% RSLogix 500 project XLT_EXP_TOP.RSS, saved by version 11.00.00.00 %
PROJECT "LINCETOP"    % processor: MicroLogix 1400 %

PROGRAM FILES
  LAD 2 "MAIN"  15 rungs  % Main Program Routine %
  LAD 70 "OFFSETS"  13 rungs
  LAD 88 "TIMESWITCH"  2 rungs
  LAD 89 "SECONDS"  2 rungs
  LAD 90 "HSC"  9 rungs
  LAD 99 "HMI SET"  3 rungs
  LAD 100 "STI"  32 rungs
  LAD 102 "SPEED"  6 rungs
  LAD 104 "P ADJUST"  8 rungs
  LAD 110 "SHIFT"  11 rungs
  LAD 120 "XFER IN"  3 rungs
  LAD 121 "NOTUSED4"  7 rungs
  LAD 122 "PARTDETECT"  9 rungs
  LAD 123 "OPTICWIDTH"  8 rungs
  LAD 124 "PART GAP"  8 rungs
  LAD 125 "NOTUSED2"  4 rungs
  LAD 126 "ALIGNLOAD"  15 rungs
  LAD 127 "NOTUSED"  3 rungs
  LAD 128 "NOTUSED3"  12 rungs
  LAD 130 "INS 5 TRIG"  30 rungs
  LAD 131 "INS 5 RSLT"  29 rungs
  LAD 140 "INS 6 TRIG"  30 rungs
  LAD 141 "INS 6 RSLT"  30 rungs
  LAD 170 "PASSBLOW"  14 rungs
  LAD 180 "RECERK"  9 rungs
  LAD 200 "PRODRATE"  6 rungs
  LAD 230 "HMI GET"  1 rungs

DATA FILES
  O0 OUTPUT  6 elements
  I1 INPUT  8 elements
  S2 STATUS  66 elements
  B3 BINARY  14 elements
  T4 TIMER  40 elements
  C5 COUNTER  1 elements
  R6 CONTROL  30 elements
  N7 INTEGER  200 elements
  F8 FLOAT  100 elements
  B9 TOP BS DAT  256 elements
  B10 TEMP  128 elements  % temp for program change %
  B11 TOP ER DAT  256 elements
  N12 TEMP  128 elements  % until sort out program io difference %
  L13  COUNTS  100 elements
  L23 NEW READ  100 elements
  L24 NEW WRITE  100 elements
  L42   52 elements
  B181 BLANK  128 elements  % used to wipe bs files %
  F182 TEST FLOAT  22 elements
  L183 TEST LONG  22 elements
  N184 TEST INTS  22 elements
  B185 TEST BITS  22 elements
  N186 HMI INTS  20 elements
  L187 HMI LONG  22 elements
  F188 HMI FLOATS  20 elements
  B189 HMI BITS  20 elements
  L190 COUNTS  128 elements
  B191 ERROR BITS  10 elements
  L192 SPD OFFSET  55 elements
  F193 SPD OFFSET  55 elements
  B194 GOOD BS  256 elements
  B195 NOERROR BS  256 elements
  B196 CTRL BITS  50 elements
  N197 CTRL INTS  50 elements
  B198 TRK BITS  50 elements
  L199 TRK LNG  50 elements
  N200 TRK INTS  50 elements
  L201 INS LNG  50 elements
  B202 INS BITS  50 elements
  N203 INS INTS  50 elements
  L204 CTRL LONG  60 elements
  F205 CTRL FLTS  50 elements

LADDER 2 "MAIN"    % Main Program Routine %
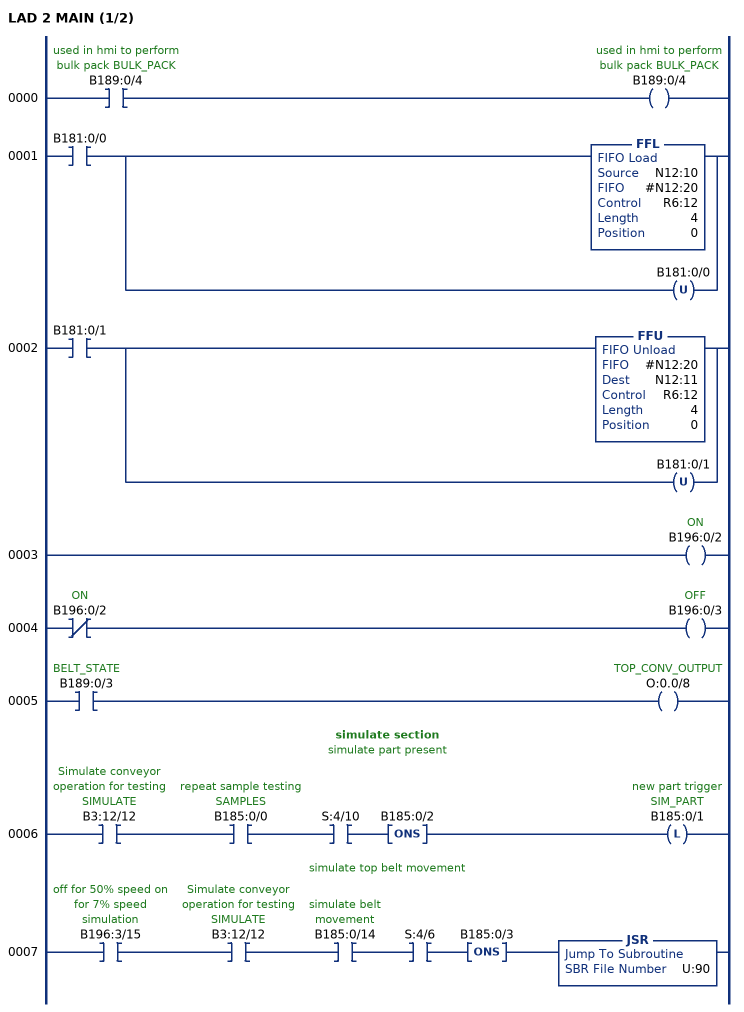
% Rung: 0 %
SOR XIC B189:0/4 OTE B189:0/4 EOR
%   B189:0/4  BULK_PACK  "used in hmi to perform bulk pack" %
% Rung: 1 %
SOR XIC B181:0/0 BST FFL N12:10 #N12:20 R6:12 4 0 NXB OTU B181:0/0 BND EOR
% Rung: 2 %
SOR XIC B181:0/1 BST FFU #N12:20 N12:11 R6:12 4 0 NXB OTU B181:0/1 BND EOR
% Rung: 3 %
SOR OTE B196:0/2 EOR
%   B196:0/2  ON %
% Rung: 4 %
SOR XIO B196:0/2 OTE B196:0/3 EOR
%   B196:0/2  ON %
%   B196:0/3  OFF %
% Rung: 5 %
SOR XIC B189:0/3 OTE O:0.0/8 EOR
%   B189:0/3  BELT_STATE %
%   O:0.0/8  TOP_CONV_OUTPUT %
% Rung: 6 %
% TITLE: simulate section %
% simulate part present %
SOR XIC B3:12/12 XIC B185:0/0 XIC S:4/10 ONS B185:0/2 OTL B185:0/1 EOR
%   B3:12/12  SIMULATE  "Simulate conveyor operation for testing" %
%   B185:0/0  SAMPLES  "repeat sample testing" %
%   B185:0/1  SIM_PART  "new part trigger" %
% Rung: 7 %
% simulate top belt movement %
SOR XIC B196:3/15 XIC B3:12/12 XIC B185:0/14 XIC S:4/6 ONS B185:0/3 JSR U:90 EOR
%   B196:3/15  "off for 50% speed on for 7% speed simulation" %
%   B3:12/12  SIMULATE  "Simulate conveyor operation for testing" %
%   B185:0/14  "simulate belt movement" %

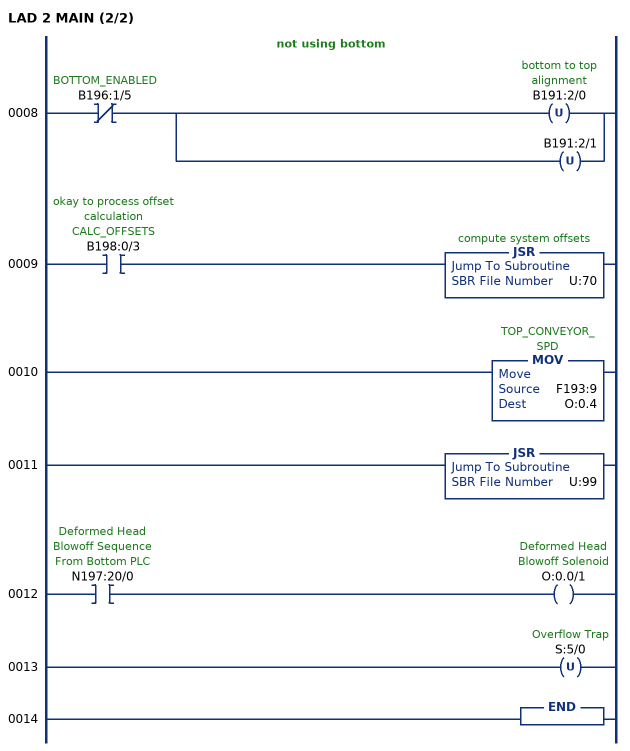
% Rung: 8 %
% TITLE: not using bottom %
SOR XIO B196:1/5 BST OTU B191:2/0 NXB OTU B191:2/1 BND EOR
%   B196:1/5  BOTTOM_ENABLED %
%   B191:2/0  "bottom to top alignment" %
% Rung: 9 %
SOR XIC B198:0/3 JSR U:70 EOR
%   B198:0/3  CALC_OFFSETS  "okay to process offset calculation" %
%   U:70  "compute system offsets" %
% Rung: 10 %
SOR MOV F193:9 O:0.4 EOR
%   F193:9  CTRLED_SCALED_VALUE %
%   O:0.4  TOP_CONVEYOR_SPD %
% Rung: 11 %
SOR JSR U:99 EOR
% Rung: 12 %
SOR XIC N197:20/0 OTE O:0.0/1 EOR
%   N197:20/0  "Deformed Head Blowoff Sequence From Bottom PLC" %
%   O:0.0/1  "Deformed Head Blowoff Solenoid" %
% Rung: 13 %
SOR OTU S:5/0 EOR
%   S:5/0  "Overflow Trap" %
% Rung: 14 %
SOR END EOR

LADDER 70 "OFFSETS"
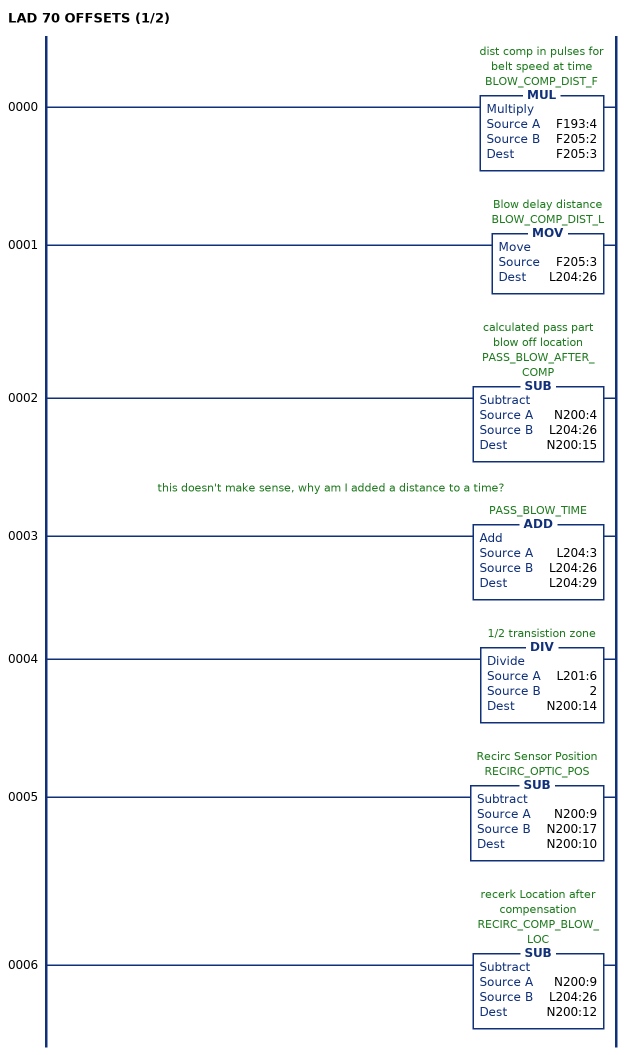
% Rung: 0 %
SOR MUL F193:4 F205:2 F205:3 EOR
%   F193:4  SCALED_SET_SPEED %
%   F205:2  BLOW_COMP_TM  "blow compensation delay time from hmi" %
%   F205:3  BLOW_COMP_DIST_F  "dist comp in pulses for belt speed at time" %
% Rung: 1 %
SOR MOV F205:3 L204:26 EOR
%   F205:3  BLOW_COMP_DIST_F  "dist comp in pulses for belt speed at time" %
%   L204:26  BLOW_COMP_DIST_L  "Blow delay distance" %
% Rung: 2 %
SOR SUB N200:4 L204:26 N200:15 EOR
%   N200:4  PASS_BLOW_LOC %
%   L204:26  BLOW_COMP_DIST_L  "Blow delay distance" %
%   N200:15  PASS_BLOW_AFTER_COMP  "calculated pass part blow off location" %
% Rung: 3 %
% this doesn't make sense, why am I added a distance to a time? %
SOR ADD L204:3 L204:26 L204:29 EOR
%   L204:3  "blow on time" %
%   L204:26  BLOW_COMP_DIST_L  "Blow delay distance" %
%   L204:29  PASS_BLOW_TIME %
% Rung: 4 %
SOR DIV L201:6 2 N200:14 EOR
%   L201:6  TRANSWINDOW  "The alignment window for the bottom to top alignment" %
%   N200:14  "1/2 transistion zone" %
% Rung: 5 %
SOR SUB N200:9 N200:17 N200:10 EOR
%   N200:9  RECIRC_BLOW_LOC %
%   N200:17  RECIRC_OFFSET  "recirc offset?" %
%   N200:10  RECIRC_OPTIC_POS  "Recirc Sensor Position" %
% Rung: 6 %
SOR SUB N200:9 L204:26 N200:12 EOR
%   N200:9  RECIRC_BLOW_LOC %
%   L204:26  BLOW_COMP_DIST_L  "Blow delay distance" %
%   N200:12  RECIRC_COMP_BLOW_LOC  "recerk Location after compensation" %

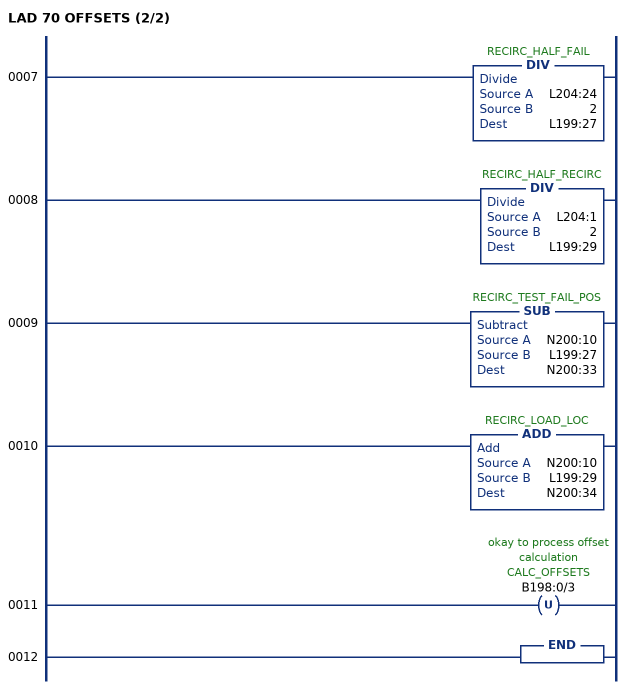
% Rung: 7 %
SOR DIV L204:24 2 L199:27 EOR
%   L204:24  RECIRC_FAIL_WINDOW  "window width" %
%   L199:27  RECIRC_HALF_FAIL %
% Rung: 8 %
SOR DIV L204:1 2 L199:29 EOR
%   L204:1  RECIRC_WINDOW %
%   L199:29  RECIRC_HALF_RECIRC %
% Rung: 9 %
SOR SUB N200:10 L199:27 N200:33 EOR
%   N200:10  RECIRC_OPTIC_POS  "Recirc Sensor Position" %
%   L199:27  RECIRC_HALF_FAIL %
%   N200:33  RECIRC_TEST_FAIL_POS %
% Rung: 10 %
SOR ADD N200:10 L199:29 N200:34 EOR
%   N200:10  RECIRC_OPTIC_POS  "Recirc Sensor Position" %
%   L199:29  RECIRC_HALF_RECIRC %
%   N200:34  RECIRC_LOAD_LOC %
% Rung: 11 %
SOR OTU B198:0/3 EOR
%   B198:0/3  CALC_OFFSETS  "okay to process offset calculation" %
% Rung: 12 %
SOR END EOR

LADDER 88 "TIMESWITCH"
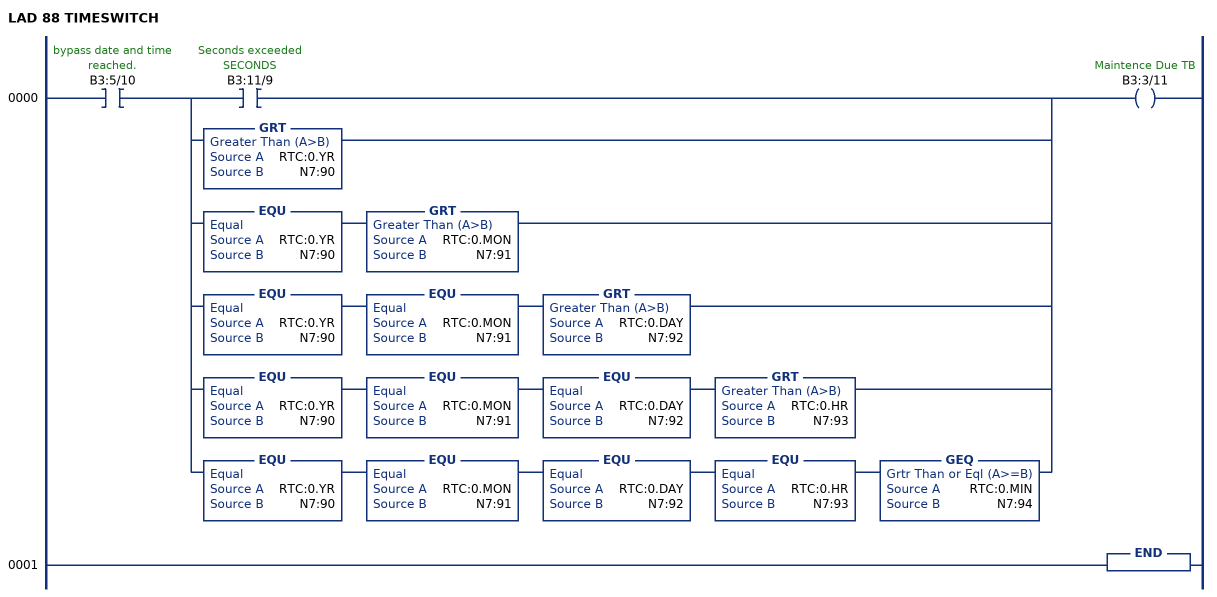
% Rung: 0 %
SOR XIC B3:5/10 BST XIC B3:11/9 NXB GRT RTC:0.YR N7:90 NXB EQU RTC:0.YR N7:90 GRT RTC:0.MON N7:91 NXB EQU RTC:0.YR N7:90 EQU RTC:0.MON N7:91 GRT RTC:0.DAY N7:92 NXB EQU RTC:0.YR N7:90 EQU RTC:0.MON N7:91 EQU RTC:0.DAY N7:92 GRT RTC:0.HR N7:93 NXB EQU RTC:0.YR N7:90 EQU RTC:0.MON N7:91 EQU RTC:0.DAY N7:92 EQU RTC:0.HR N7:93 GEQ RTC:0.MIN N7:94 BND OTE B3:3/11 EOR
%   B3:5/10  "bypass date and time reached." %
%   B3:11/9  SECONDS  "Seconds exceeded" %
%   N7:90  RTC %
%   B3:3/11  TB  "Maintence Due" %
% Rung: 1 %
SOR END EOR

LADDER 89 "SECONDS"
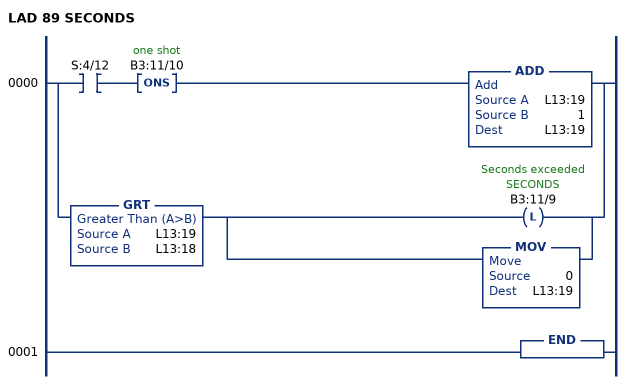
% Rung: 0 %
SOR BST XIC S:4/12 ONS B3:11/10 ADD L13:19 1 L13:19 NXB GRT L13:19 L13:18 BST OTL B3:11/9 NXB MOV 0 L13:19 BND BND EOR
%   B3:11/10  "one shot" %
%   L13:18  MAX %
%   B3:11/9  SECONDS  "Seconds exceeded" %
% Rung: 1 %
SOR END EOR

LADDER 90 "HSC"
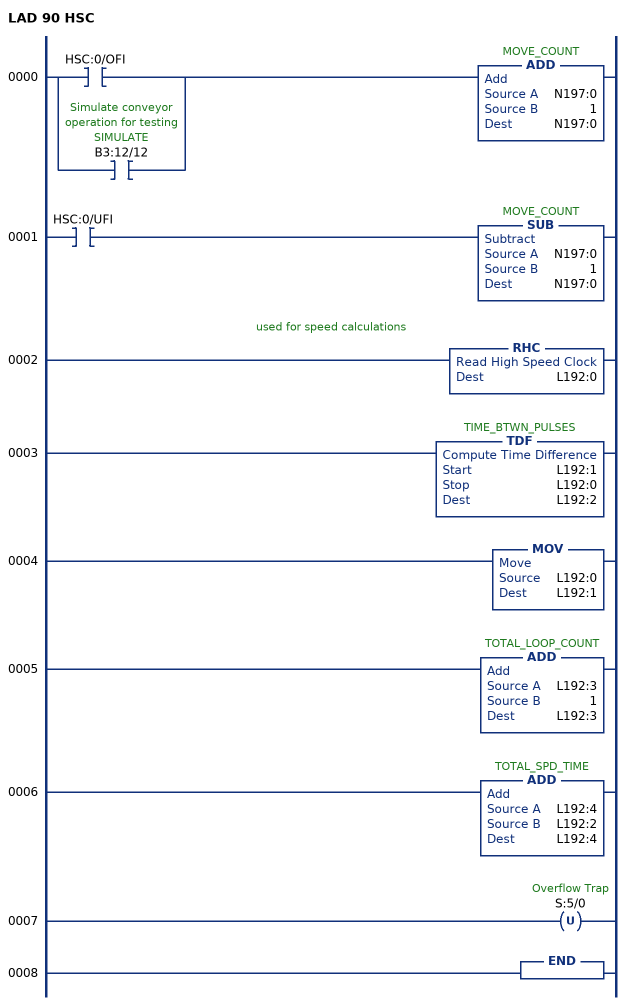
% Rung: 0 %
SOR BST XIC HSC:0/OFI NXB XIC B3:12/12 BND ADD N197:0 1 N197:0 EOR
%   B3:12/12  SIMULATE  "Simulate conveyor operation for testing" %
%   N197:0  MOVE_COUNT %
% Rung: 1 %
SOR XIC HSC:0/UFI SUB N197:0 1 N197:0 EOR
%   N197:0  MOVE_COUNT %
% Rung: 2 %
% used for speed calculations %
SOR RHC L192:0 EOR
% Rung: 3 %
SOR TDF L192:1 L192:0 L192:2 EOR
%   L192:2  TIME_BTWN_PULSES %
% Rung: 4 %
SOR MOV L192:0 L192:1 EOR
% Rung: 5 %
SOR ADD L192:3 1 L192:3 EOR
%   L192:3  TOTAL_LOOP_COUNT %
% Rung: 6 %
SOR ADD L192:4 L192:2 L192:4 EOR
%   L192:4  TOTAL_SPD_TIME %
%   L192:2  TIME_BTWN_PULSES %
% Rung: 7 %
SOR OTU S:5/0 EOR
%   S:5/0  "Overflow Trap" %
% Rung: 8 %
SOR END EOR

LADDER 99 "HMI SET"
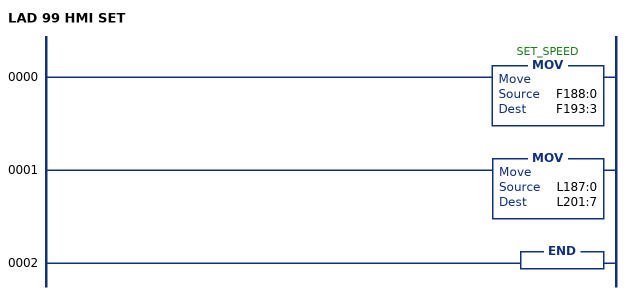
% Rung: 0 %
SOR MOV F188:0 F193:3 EOR
%   F188:0  HMI_SPEED  "hmi belt speed setting input" %
%   F193:3  SET_SPEED %
% Rung: 1 %
SOR MOV L187:0 L201:7 EOR
%   L187:0  ALIGN_OFFSET_MIN %
% Rung: 2 %
SOR END EOR

LADDER 100 "STI"
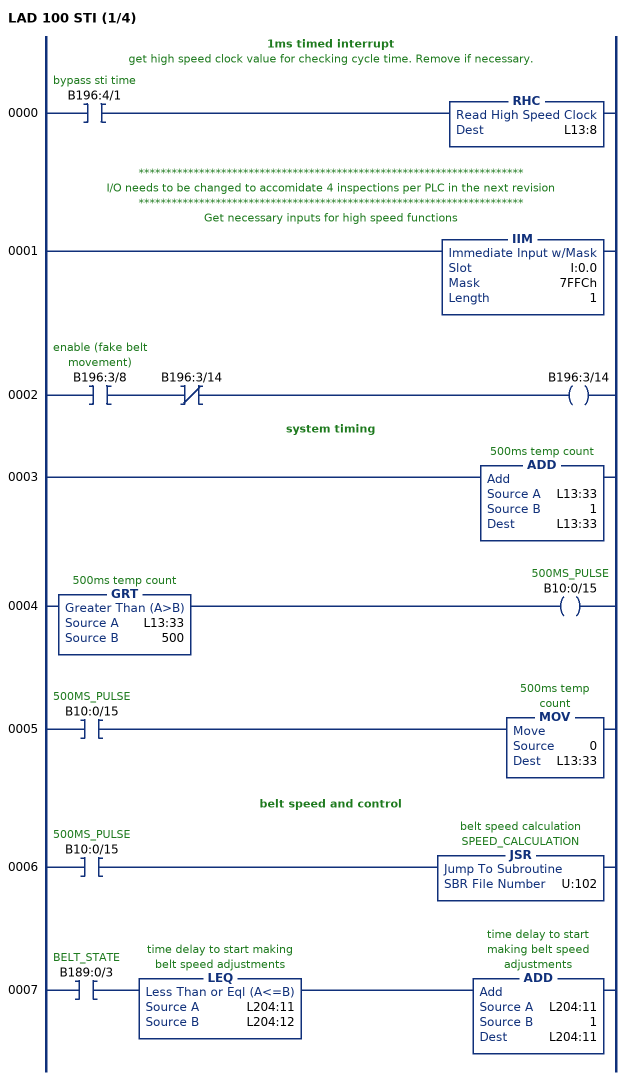
% Rung: 0 %
% TITLE: 1ms timed interrupt %
% get high speed clock value for checking cycle time. Remove if necessary. %
SOR XIC B196:4/1 RHC L13:8 EOR
%   B196:4/1  "bypass sti time" %
% Rung: 1 %
% **********************************************************************
% 
% I/O needs to be changed to accomidate 4 inspections per PLC in the next revision
% 
% **********************************************************************
% 
% Get necessary inputs for high speed functions %
SOR IIM I:0.0 7FFCh 1 EOR
% Rung: 2 %
SOR XIC B196:3/8 XIO B196:3/14 OTE B196:3/14 EOR
%   B196:3/8  "enable (fake belt movement)" %
% Rung: 3 %
% TITLE: system timing %
SOR ADD L13:33 1 L13:33 EOR
%   L13:33  "500ms temp count" %
% Rung: 4 %
SOR GRT L13:33 500 OTE B10:0/15 EOR
%   L13:33  "500ms temp count" %
%   B10:0/15  500MS_PULSE %
% Rung: 5 %
SOR XIC B10:0/15 MOV 0 L13:33 EOR
%   B10:0/15  500MS_PULSE %
%   L13:33  "500ms temp count" %
% Rung: 6 %
% TITLE: belt speed and control %
SOR XIC B10:0/15 JSR U:102 EOR
%   B10:0/15  500MS_PULSE %
%   U:102  SPEED_CALCULATION  "belt speed calculation" %
% Rung: 7 %
SOR XIC B189:0/3 LEQ L204:11 L204:12 ADD L204:11 1 L204:11 EOR
%   B189:0/3  BELT_STATE %
%   L204:11  "time delay to start making belt speed adjustments" %

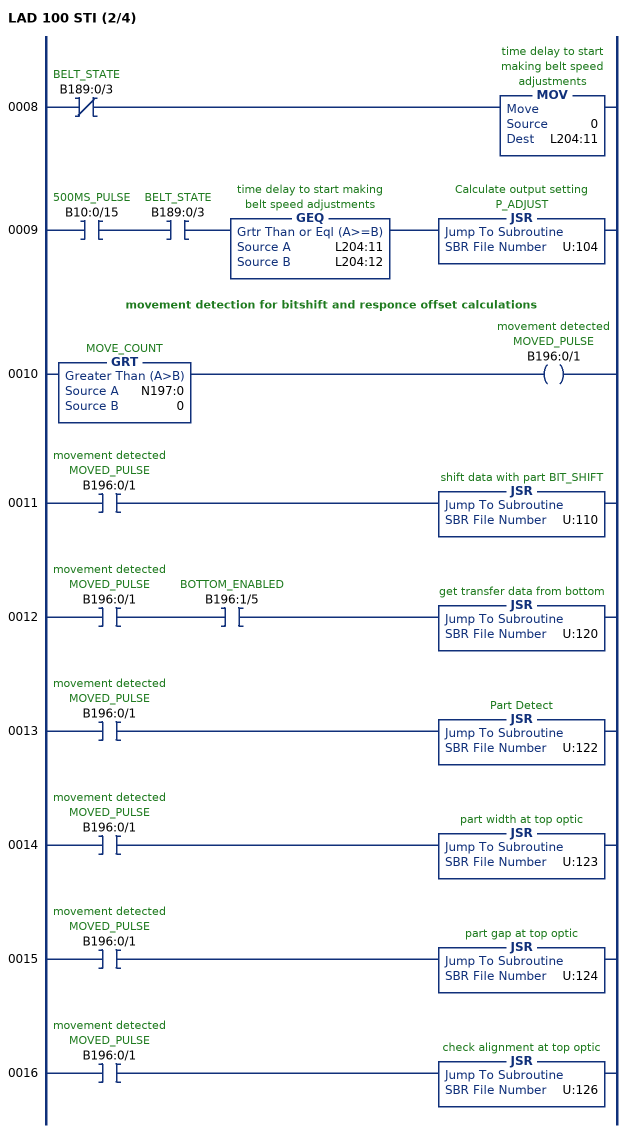
% Rung: 8 %
SOR XIO B189:0/3 MOV 0 L204:11 EOR
%   B189:0/3  BELT_STATE %
%   L204:11  "time delay to start making belt speed adjustments" %
% Rung: 9 %
SOR XIC B10:0/15 XIC B189:0/3 GEQ L204:11 L204:12 JSR U:104 EOR
%   B10:0/15  500MS_PULSE %
%   B189:0/3  BELT_STATE %
%   L204:11  "time delay to start making belt speed adjustments" %
%   U:104  P_ADJUST  "Calculate output setting" %
% Rung: 10 %
% TITLE: movement detection for bitshift and responce offset calculations %
SOR GRT N197:0 0 OTE B196:0/1 EOR
%   N197:0  MOVE_COUNT %
%   B196:0/1  MOVED_PULSE  "movement detected" %
% Rung: 11 %
SOR XIC B196:0/1 JSR U:110 EOR
%   B196:0/1  MOVED_PULSE  "movement detected" %
%   U:110  BIT_SHIFT  "shift data with part" %
% Rung: 12 %
SOR XIC B196:0/1 XIC B196:1/5 JSR U:120 EOR
%   B196:0/1  MOVED_PULSE  "movement detected" %
%   B196:1/5  BOTTOM_ENABLED %
%   U:120  "get transfer data from bottom" %
% Rung: 13 %
SOR XIC B196:0/1 JSR U:122 EOR
%   B196:0/1  MOVED_PULSE  "movement detected" %
%   U:122  "Part Detect" %
% Rung: 14 %
SOR XIC B196:0/1 JSR U:123 EOR
%   B196:0/1  MOVED_PULSE  "movement detected" %
%   U:123  "part width at top optic" %
% Rung: 15 %
SOR XIC B196:0/1 JSR U:124 EOR
%   B196:0/1  MOVED_PULSE  "movement detected" %
%   U:124  "part gap at top optic" %
% Rung: 16 %
SOR XIC B196:0/1 JSR U:126 EOR
%   B196:0/1  MOVED_PULSE  "movement detected" %
%   U:126  "check alignment at top optic" %

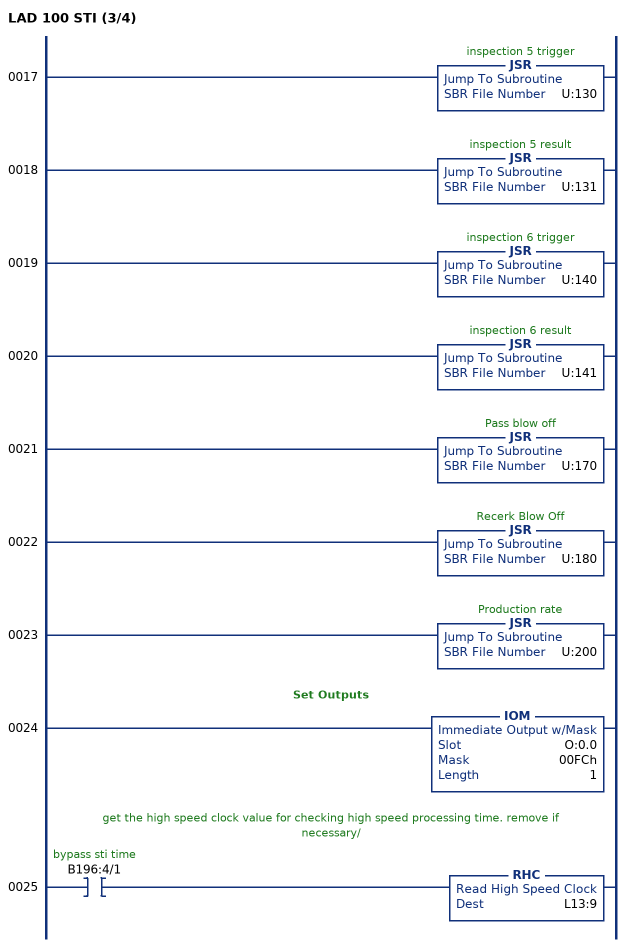
% Rung: 17 %
SOR JSR U:130 EOR
%   U:130  "inspection 5 trigger" %
% Rung: 18 %
SOR JSR U:131 EOR
%   U:131  "inspection 5 result" %
% Rung: 19 %
SOR JSR U:140 EOR
%   U:140  "inspection 6 trigger" %
% Rung: 20 %
SOR JSR U:141 EOR
%   U:141  "inspection 6 result" %
% Rung: 21 %
SOR JSR U:170 EOR
%   U:170  "Pass blow off" %
% Rung: 22 %
SOR JSR U:180 EOR
%   U:180  "Recerk Blow Off" %
% Rung: 23 %
SOR JSR U:200 EOR
%   U:200  "Production rate" %
% Rung: 24 %
% TITLE: Set Outputs %
SOR IOM O:0.0 00FCh 1 EOR
% Rung: 25 %
% get the high speed clock value for checking high speed processing time. remove if necessary/ %
SOR XIC B196:4/1 RHC L13:9 EOR
%   B196:4/1  "bypass sti time" %

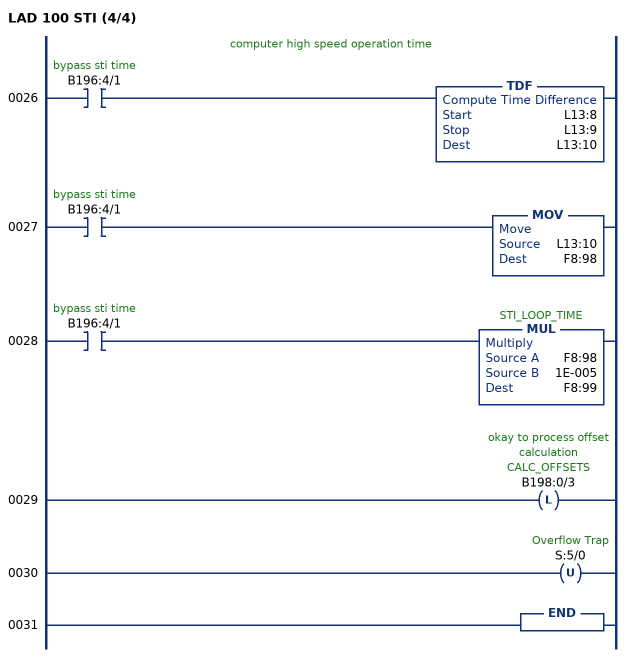
% Rung: 26 %
% computer high speed operation time %
SOR XIC B196:4/1 TDF L13:8 L13:9 L13:10 EOR
%   B196:4/1  "bypass sti time" %
% Rung: 27 %
SOR XIC B196:4/1 MOV L13:10 F8:98 EOR
%   B196:4/1  "bypass sti time" %
% Rung: 28 %
SOR XIC B196:4/1 MUL F8:98 1E-005 F8:99 EOR
%   B196:4/1  "bypass sti time" %
%   F8:99  STI_LOOP_TIME %
% Rung: 29 %
SOR OTL B198:0/3 EOR
%   B198:0/3  CALC_OFFSETS  "okay to process offset calculation" %
% Rung: 30 %
SOR OTU S:5/0 EOR
%   S:5/0  "Overflow Trap" %
% Rung: 31 %
SOR END EOR

LADDER 102 "SPEED"
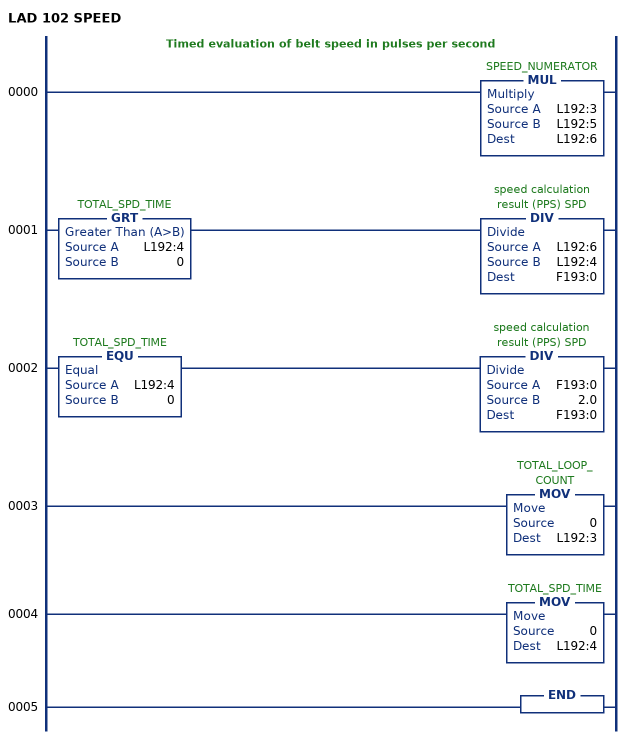
% Rung: 0 %
% TITLE: Timed evaluation of belt speed in pulses per second %
SOR MUL L192:3 L192:5 L192:6 EOR
%   L192:3  TOTAL_LOOP_COUNT %
%   L192:5  TKS_PER_SECOND %
%   L192:6  SPEED_NUMERATOR %
% Rung: 1 %
SOR GRT L192:4 0 DIV L192:6 L192:4 F193:0 EOR
%   L192:4  TOTAL_SPD_TIME %
%   L192:6  SPEED_NUMERATOR %
%   F193:0  SPD  "speed calculation result (PPS)" %
% Rung: 2 %
SOR EQU L192:4 0 DIV F193:0 2.0 F193:0 EOR
%   L192:4  TOTAL_SPD_TIME %
%   F193:0  SPD  "speed calculation result (PPS)" %
% Rung: 3 %
SOR MOV 0 L192:3 EOR
%   L192:3  TOTAL_LOOP_COUNT %
% Rung: 4 %
SOR MOV 0 L192:4 EOR
%   L192:4  TOTAL_SPD_TIME %
% Rung: 5 %
SOR END EOR

LADDER 104 "P ADJUST"
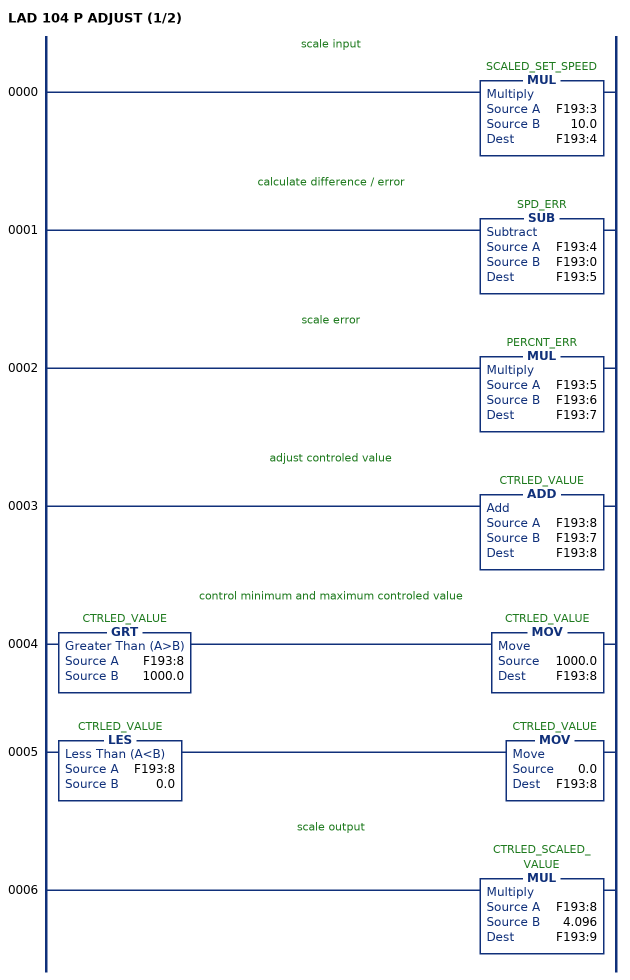
% Rung: 0 %
% scale input %
SOR MUL F193:3 10.0 F193:4 EOR
%   F193:3  SET_SPEED %
%   F193:4  SCALED_SET_SPEED %
% Rung: 1 %
% calculate difference / error %
SOR SUB F193:4 F193:0 F193:5 EOR
%   F193:4  SCALED_SET_SPEED %
%   F193:0  SPD  "speed calculation result (PPS)" %
%   F193:5  SPD_ERR %
% Rung: 2 %
% scale error %
SOR MUL F193:5 F193:6 F193:7 EOR
%   F193:5  SPD_ERR %
%   F193:6  FDBK_RATIO %
%   F193:7  PERCNT_ERR %
% Rung: 3 %
% adjust controled value %
SOR ADD F193:8 F193:7 F193:8 EOR
%   F193:8  CTRLED_VALUE %
%   F193:7  PERCNT_ERR %
% Rung: 4 %
% control minimum and maximum controled value %
SOR GRT F193:8 1000.0 MOV 1000.0 F193:8 EOR
%   F193:8  CTRLED_VALUE %
% Rung: 5 %
SOR LES F193:8 0.0 MOV 0.0 F193:8 EOR
%   F193:8  CTRLED_VALUE %
% Rung: 6 %
% scale output %
SOR MUL F193:8 4.096 F193:9 EOR
%   F193:8  CTRLED_VALUE %
%   F193:9  CTRLED_SCALED_VALUE %

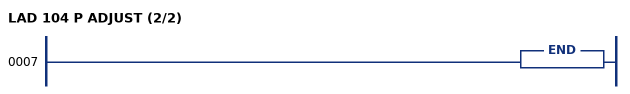
% Rung: 7 %
SOR END EOR

LADDER 110 "SHIFT"
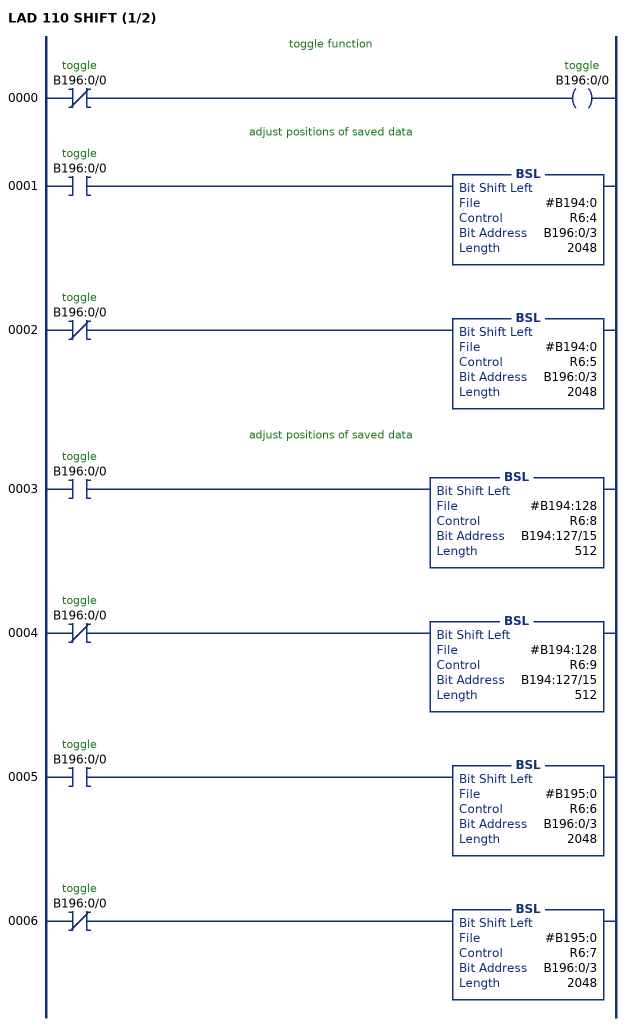
% Rung: 0 %
% toggle function %
SOR XIO B196:0/0 OTE B196:0/0 EOR
%   B196:0/0  "toggle" %
% Rung: 1 %
% adjust positions of saved data %
SOR XIC B196:0/0 BSL #B194:0 R6:4 B196:0/3 2048 EOR
%   B196:0/0  "toggle" %
%   B196:0/3  OFF %
% Rung: 2 %
SOR XIO B196:0/0 BSL #B194:0 R6:5 B196:0/3 2048 EOR
%   B196:0/0  "toggle" %
%   B196:0/3  OFF %
% Rung: 3 %
% adjust positions of saved data %
SOR XIC B196:0/0 BSL #B194:128 R6:8 B194:127/15 512 EOR
%   B196:0/0  "toggle" %
% Rung: 4 %
SOR XIO B196:0/0 BSL #B194:128 R6:9 B194:127/15 512 EOR
%   B196:0/0  "toggle" %
% Rung: 5 %
SOR XIC B196:0/0 BSL #B195:0 R6:6 B196:0/3 2048 EOR
%   B196:0/0  "toggle" %
%   B196:0/3  OFF %
% Rung: 6 %
SOR XIO B196:0/0 BSL #B195:0 R6:7 B196:0/3 2048 EOR
%   B196:0/0  "toggle" %
%   B196:0/3  OFF %

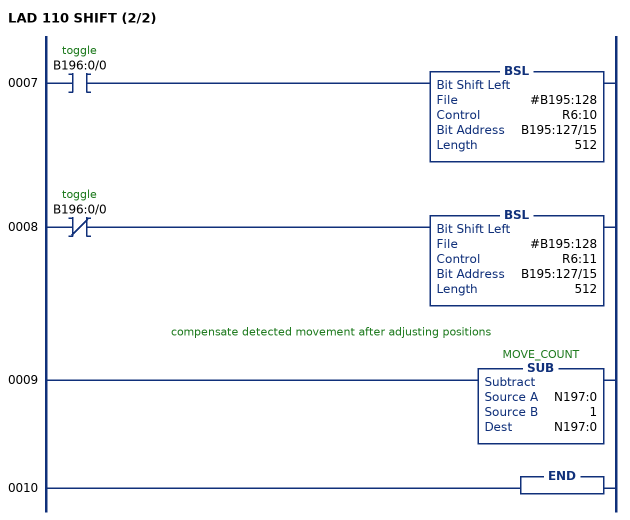
% Rung: 7 %
SOR XIC B196:0/0 BSL #B195:128 R6:10 B195:127/15 512 EOR
%   B196:0/0  "toggle" %
% Rung: 8 %
SOR XIO B196:0/0 BSL #B195:128 R6:11 B195:127/15 512 EOR
%   B196:0/0  "toggle" %
% Rung: 9 %
% compensate detected movement after adjusting positions %
SOR SUB N197:0 1 N197:0 EOR
%   N197:0  MOVE_COUNT %
% Rung: 10 %
SOR END EOR

LADDER 120 "XFER IN"
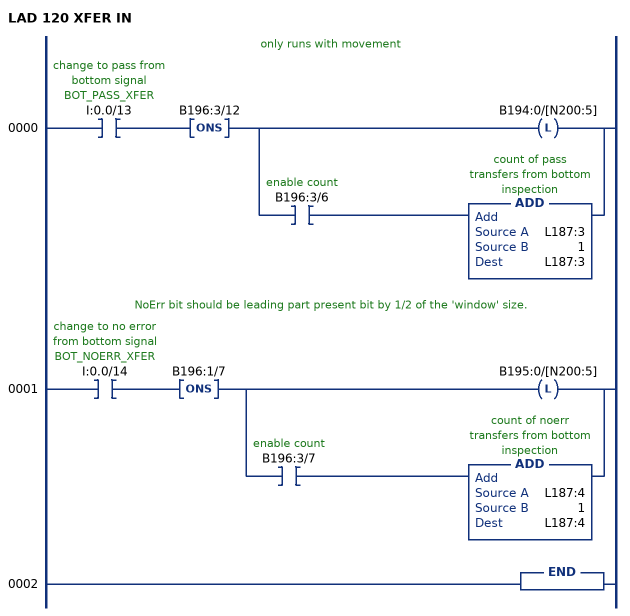
% Rung: 0 %
% only runs with movement %
SOR XIC I:0.0/13 ONS B196:3/12 BST OTL B194:0/[N200:5] NXB XIC B196:3/6 ADD L187:3 1 L187:3 BND EOR
%   I:0.0/13  BOT_PASS_XFER  "change to pass from bottom signal" %
%   N200:5  TOP_LOAD %
%   B196:3/6  "enable count" %
%   L187:3  "count of pass transfers from bottom inspection" %
% Rung: 1 %
% NoErr bit should be leading part present bit by 1/2 of the 'window' size. %
SOR XIC I:0.0/14 ONS B196:1/7 BST OTL B195:0/[N200:5] NXB XIC B196:3/7 ADD L187:4 1 L187:4 BND EOR
%   I:0.0/14  BOT_NOERR_XFER  "change to no error from bottom signal" %
%   N200:5  TOP_LOAD %
%   B196:3/7  "enable count" %
%   L187:4  "count of noerr transfers from bottom inspection" %
% Rung: 2 %
SOR END EOR

LADDER 121 "NOTUSED4"
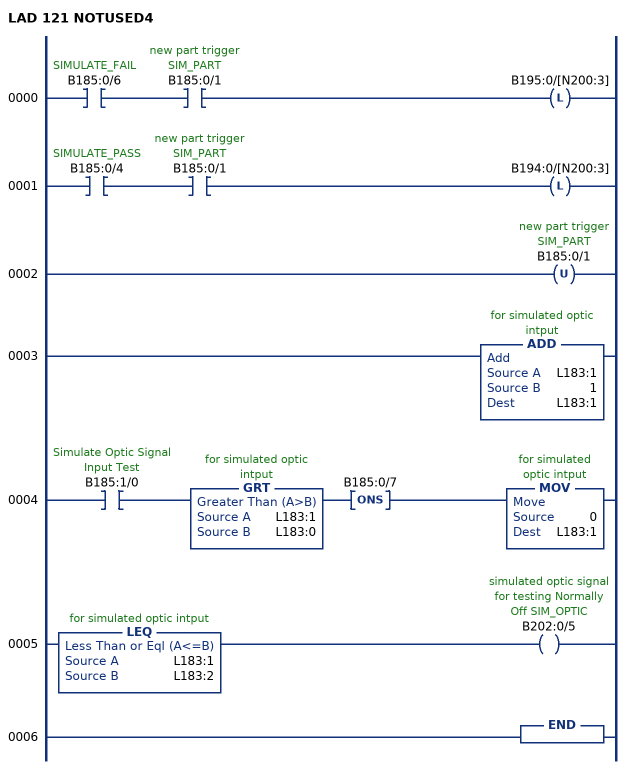
% Rung: 0 %
SOR XIC B185:0/6 XIC B185:0/1 OTL B195:0/[N200:3] EOR
%   B185:0/6  SIMULATE_FAIL %
%   B185:0/1  SIM_PART  "new part trigger" %
%   N200:3  OPT_LD_PT %
% Rung: 1 %
SOR XIC B185:0/4 XIC B185:0/1 OTL B194:0/[N200:3] EOR
%   B185:0/4  SIMULATE_PASS %
%   B185:0/1  SIM_PART  "new part trigger" %
%   N200:3  OPT_LD_PT %
% Rung: 2 %
SOR OTU B185:0/1 EOR
%   B185:0/1  SIM_PART  "new part trigger" %
% Rung: 3 %
SOR ADD L183:1 1 L183:1 EOR
%   L183:1  "for simulated optic intput" %
% Rung: 4 %
SOR XIC B185:1/0 GRT L183:1 L183:0 ONS B185:0/7 MOV 0 L183:1 EOR
%   B185:1/0  "Simulate Optic Signal Input Test" %
%   L183:1  "for simulated optic intput" %
%   L183:0  "Movement pulse count for part data injection" %
% Rung: 5 %
SOR LEQ L183:1 L183:2 OTE B202:0/5 EOR
%   L183:1  "for simulated optic intput" %
%   L183:2  "simulated part width" %
%   B202:0/5  SIM_OPTIC  "simulated optic signal for testing Normally Off" %
% Rung: 6 %
SOR END EOR

LADDER 122 "PARTDETECT"
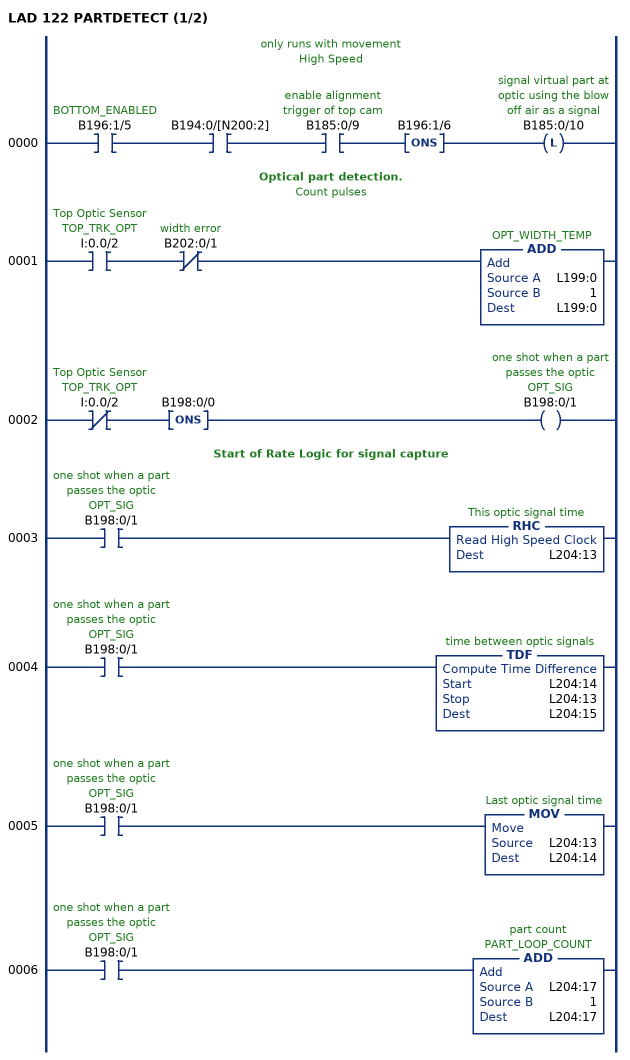
% Rung: 0 %
% only runs with movement
% High Speed %
SOR XIC B196:1/5 XIC B194:0/[N200:2] XIC B185:0/9 ONS B196:1/6 OTL B185:0/10 EOR
%   B196:1/5  BOTTOM_ENABLED %
%   N200:2  OPTIC_LOC  "top optic location" %
%   B185:0/9  "enable alignment trigger of top cam" %
%   B185:0/10  "signal virtual part at optic using the blow off air as a signal" %
% Rung: 1 %
% TITLE: Optical part detection. %
% Count pulses %
SOR XIC I:0.0/2 XIO B202:0/1 ADD L199:0 1 L199:0 EOR
%   I:0.0/2  TOP_TRK_OPT  "Top Optic Sensor" %
%   B202:0/1  "width error" %
%   L199:0  OPT_WIDTH_TEMP %
% Rung: 2 %
SOR XIO I:0.0/2 ONS B198:0/0 OTE B198:0/1 EOR
%   I:0.0/2  TOP_TRK_OPT  "Top Optic Sensor" %
%   B198:0/1  OPT_SIG  "one shot when a part passes the optic" %
% Rung: 3 %
% TITLE: Start of Rate Logic for signal capture %
SOR XIC B198:0/1 RHC L204:13 EOR
%   B198:0/1  OPT_SIG  "one shot when a part passes the optic" %
%   L204:13  "This optic signal time" %
% Rung: 4 %
SOR XIC B198:0/1 TDF L204:14 L204:13 L204:15 EOR
%   B198:0/1  OPT_SIG  "one shot when a part passes the optic" %
%   L204:14  "Last optic signal time" %
%   L204:13  "This optic signal time" %
%   L204:15  "time between optic signals" %
% Rung: 5 %
SOR XIC B198:0/1 MOV L204:13 L204:14 EOR
%   B198:0/1  OPT_SIG  "one shot when a part passes the optic" %
%   L204:13  "This optic signal time" %
%   L204:14  "Last optic signal time" %
% Rung: 6 %
SOR XIC B198:0/1 ADD L204:17 1 L204:17 EOR
%   B198:0/1  OPT_SIG  "one shot when a part passes the optic" %
%   L204:17  PART_LOOP_COUNT  "part count" %

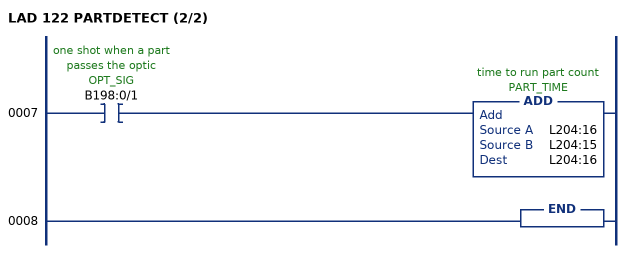
% Rung: 7 %
SOR XIC B198:0/1 ADD L204:16 L204:15 L204:16 EOR
%   B198:0/1  OPT_SIG  "one shot when a part passes the optic" %
%   L204:16  PART_TIME  "time to run part count" %
%   L204:15  "time between optic signals" %
% Rung: 8 %
SOR END EOR

LADDER 123 "OPTICWIDTH"
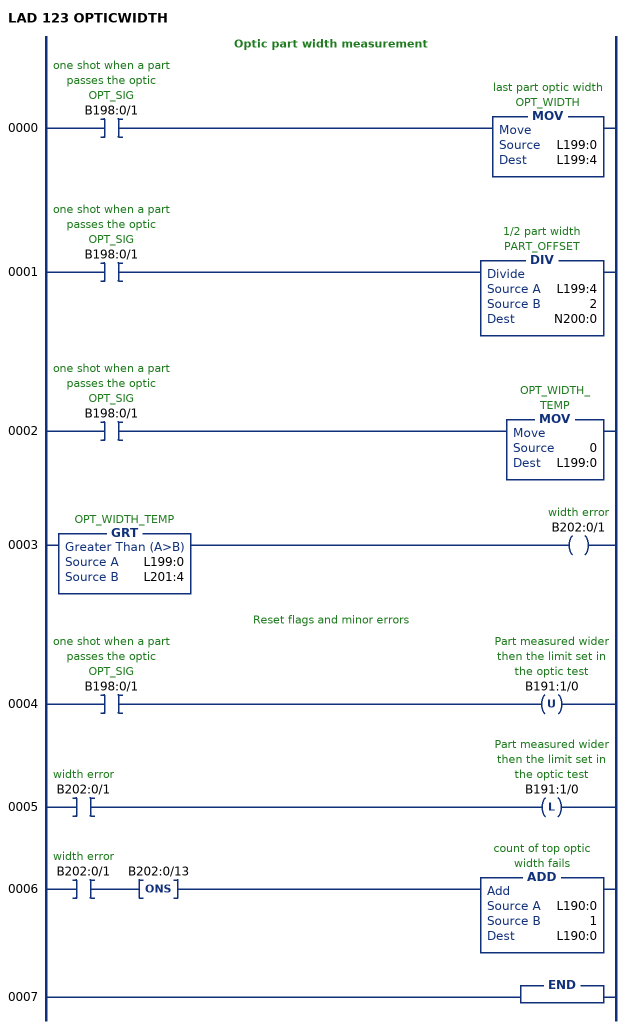
% Rung: 0 %
% TITLE: Optic part width measurement %
SOR XIC B198:0/1 MOV L199:0 L199:4 EOR
%   B198:0/1  OPT_SIG  "one shot when a part passes the optic" %
%   L199:0  OPT_WIDTH_TEMP %
%   L199:4  OPT_WIDTH  "last part optic width" %
% Rung: 1 %
SOR XIC B198:0/1 DIV L199:4 2 N200:0 EOR
%   B198:0/1  OPT_SIG  "one shot when a part passes the optic" %
%   L199:4  OPT_WIDTH  "last part optic width" %
%   N200:0  PART_OFFSET  "1/2 part width" %
% Rung: 2 %
SOR XIC B198:0/1 MOV 0 L199:0 EOR
%   B198:0/1  OPT_SIG  "one shot when a part passes the optic" %
%   L199:0  OPT_WIDTH_TEMP %
% Rung: 3 %
SOR GRT L199:0 L201:4 OTE B202:0/1 EOR
%   L199:0  OPT_WIDTH_TEMP %
%   L201:4  MAX_WIDTH  "hmi in" %
%   B202:0/1  "width error" %
% Rung: 4 %
% Reset flags and minor errors %
SOR XIC B198:0/1 OTU B191:1/0 EOR
%   B198:0/1  OPT_SIG  "one shot when a part passes the optic" %
%   B191:1/0  "Part measured wider then the limit set in the optic test" %
% Rung: 5 %
SOR XIC B202:0/1 OTL B191:1/0 EOR
%   B202:0/1  "width error" %
%   B191:1/0  "Part measured wider then the limit set in the optic test" %
% Rung: 6 %
SOR XIC B202:0/1 ONS B202:0/13 ADD L190:0 1 L190:0 EOR
%   B202:0/1  "width error" %
%   L190:0  "count of top optic width fails" %
% Rung: 7 %
SOR END EOR

LADDER 124 "PART GAP"
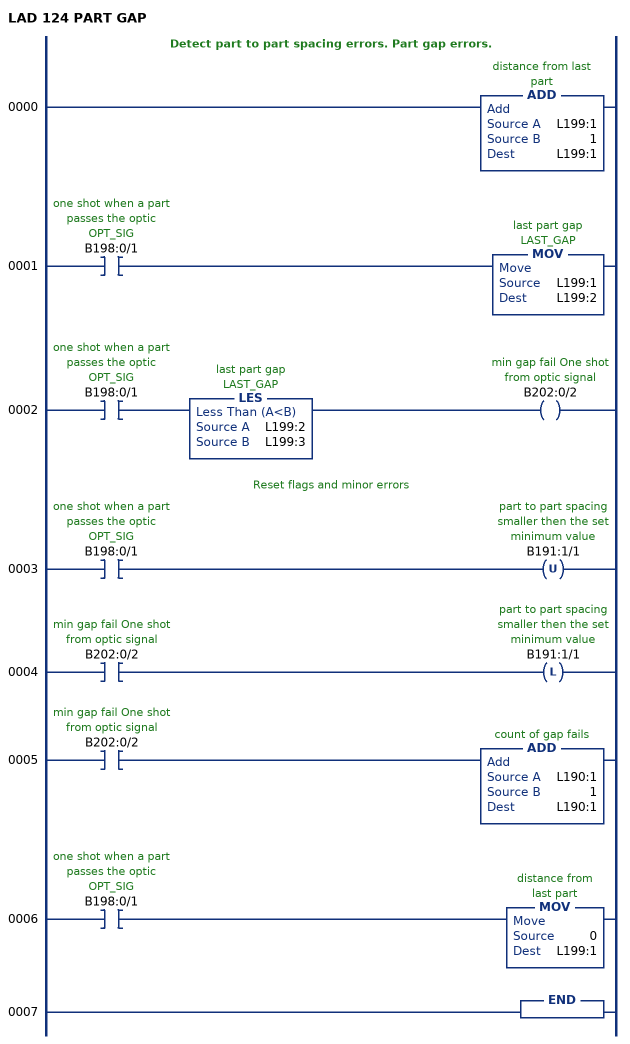
% Rung: 0 %
% TITLE: Detect part to part spacing errors. Part gap errors. %
SOR ADD L199:1 1 L199:1 EOR
%   L199:1  "distance from last part" %
% Rung: 1 %
SOR XIC B198:0/1 MOV L199:1 L199:2 EOR
%   B198:0/1  OPT_SIG  "one shot when a part passes the optic" %
%   L199:1  "distance from last part" %
%   L199:2  LAST_GAP  "last part gap" %
% Rung: 2 %
SOR XIC B198:0/1 LES L199:2 L199:3 OTE B202:0/2 EOR
%   B198:0/1  OPT_SIG  "one shot when a part passes the optic" %
%   L199:2  LAST_GAP  "last part gap" %
%   L199:3  MIN_WIDTH %
%   B202:0/2  "min gap fail One shot from optic signal" %
% Rung: 3 %
% Reset flags and minor errors %
SOR XIC B198:0/1 OTU B191:1/1 EOR
%   B198:0/1  OPT_SIG  "one shot when a part passes the optic" %
%   B191:1/1  "part to part spacing smaller then the set minimum value" %
% Rung: 4 %
SOR XIC B202:0/2 OTL B191:1/1 EOR
%   B202:0/2  "min gap fail One shot from optic signal" %
%   B191:1/1  "part to part spacing smaller then the set minimum value" %
% Rung: 5 %
SOR XIC B202:0/2 ADD L190:1 1 L190:1 EOR
%   B202:0/2  "min gap fail One shot from optic signal" %
%   L190:1  "count of gap fails" %
% Rung: 6 %
SOR XIC B198:0/1 MOV 0 L199:1 EOR
%   B198:0/1  OPT_SIG  "one shot when a part passes the optic" %
%   L199:1  "distance from last part" %
% Rung: 7 %
SOR END EOR

LADDER 125 "NOTUSED2"
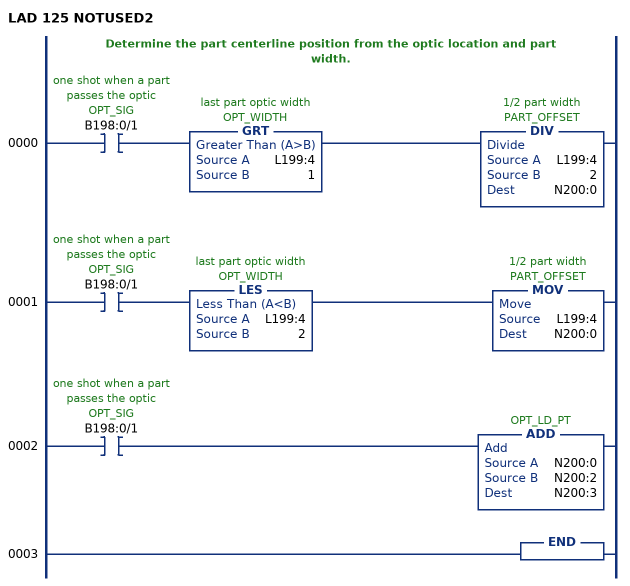
% Rung: 0 %
% TITLE: Determine the part centerline position from the optic location and part width. %
SOR XIC B198:0/1 GRT L199:4 1 DIV L199:4 2 N200:0 EOR
%   B198:0/1  OPT_SIG  "one shot when a part passes the optic" %
%   L199:4  OPT_WIDTH  "last part optic width" %
%   N200:0  PART_OFFSET  "1/2 part width" %
% Rung: 1 %
SOR XIC B198:0/1 LES L199:4 2 MOV L199:4 N200:0 EOR
%   B198:0/1  OPT_SIG  "one shot when a part passes the optic" %
%   L199:4  OPT_WIDTH  "last part optic width" %
%   N200:0  PART_OFFSET  "1/2 part width" %
% Rung: 2 %
SOR XIC B198:0/1 ADD N200:0 N200:2 N200:3 EOR
%   B198:0/1  OPT_SIG  "one shot when a part passes the optic" %
%   N200:0  PART_OFFSET  "1/2 part width" %
%   N200:2  OPTIC_LOC  "top optic location" %
%   N200:3  OPT_LD_PT %
% Rung: 3 %
SOR END EOR

LADDER 126 "ALIGNLOAD"
